Universal Robots PolyScope program: rtdeCommanding.urp

Program rtdeCommanding (installation=default directory=/programs/RemoteOperation createdIn=3.2.19275.0 lastSavedIn=5.10.0.106268 robotSerialNumber=20185500191)
Calibrated DH parameters: a=[0.000131, -0.165639, -0.102041, 0.000082, 0.000046, 0]; d=[0.162455, 220.258006, 1988.136334, -2208.260978, 0.099826, 0.099896]; alpha=[1.570482, -0.001777, -0.000172, 1.570393, -1.570735, 0]; deltaTheta=[0, -1.170526, -0.137148, 1.307669, -0.000001, 0]
BeforeStart
  setq := get_actual_joint_positions()
  servoing := 0
  SuppressedNode
    Script: rtde_set_watchdog("input_integer_register_1", 500, "pause")
Robot Program (runOnlyOnce=true)
  Script: write_output_integer_register(0, 0)
  Script: sync()
  MoveJ speed 60 deg/s, acceleration 80 deg/s^2 (useActiveTCP=true) feature=Base
    Waypoint Waypoint_1: TCP in base x=66.896 y=-541.762 z=407.404 mm, rx=2.1914 ry=2.251 rz=0 rad; joints [-68.794, -96.625, -69.102, -104.272, 89.916, 109.668] deg; TCP offset x=0 y=0 z=174 mm, rx=0 ry=0 rz=0 rad
  Script: write_output_integer_register(0, 1)
  Loop While (checkContinuously=false) expression=servoing≠1
    Script: sync()
  Loop While (checkContinuously=false) expression=servoing≟1
    Script: servoj(setq, t=0.002)
  Script: stopj(2)
  Script: write_output_integer_register(0, 0)
  Script: sync()
Thread Thread_1 (runOnlyOnce=false)
  Folder Registers
    tmp := [0.,0,0,0,0,0]
    Script: tmp[0] = read_input_float_register(0)
    Script: tmp[1] = read_input_float_register(1)
    Script: tmp[2] = read_input_float_register(2)
    Script: tmp[3] = read_input_float_register(3)
    Script: tmp[4] = read_input_float_register(4)
    Script: tmp[5] = read_input_float_register(5)
    If tmp != [0,0,0,0,0,0]
      setq := tmp
  Script: sync()
Thread Thread_2 (runOnlyOnce=false)
  servoing := read_input_integer_register(0)
  Script: sync()
